FUNCTION_BLOCK FB_trajBase
VAR_INPUT
END_VAR
VAR_OUTPUT
END_VAR
VAR
	// total trajectory duration
	m_duration :LREAL:=0;
	
	// flag is trajectory is init successfully 
	m_isGenerated : BOOL :=FALSE;
END_VAR

PROPERTY duration : lreal
GET
duration:=m_duration;
END_GET
END_PROPERTY

PROPERTY isGene : bool
GET
isGene:=m_isGenerated;
END_GET
END_PROPERTY

END_FUNCTION_BLOCK

(* stored: Version 1.1.0.1, ProductVersion 3.1.4024.12
   POU FB_trajBase: Id {f82b2b7b-78c8-43b3-8920-9f856daa52d8}, SpecialFunc None
   Property duration: Id {b4ade5b1-eaa6-4e50-b5ce-32104382721a}
   Get Get: Id {606bb1de-0742-4a23-914c-c42332aad377}
   Property isGene: Id {749168c0-621a-4da1-936e-d65a95c2edeb}
   Get Get: Id {14e08cf2-4a1a-4960-8b51-b97817f37afb} *)
